FUNCTION_BLOCK Scanner_FB
VAR_INPUT
	mxEnable: BOOL;
	mxRP: BOOL;
	mxYP: BOOL;
	mxBP: BOOL;
	mxRCy: BOOL;
	mxYCy: BOOL;
	mxBCy: BOOL;
	mxYOct: BOOL;
	mxBOct: BOOL;
	mxROct: BOOL;
	mxIP: BOOL;
	mxRCon: BOOL;
	mxYCon: BOOL;
	mxBCon: BOOL;
END_VAR
VAR_OUTPUT
	
END_VAR
VAR
	TASK: INT;
	qxScanBuffer_1:BOOL;
	qxScanBuffer_2:BOOL;
	qxScanBuffer_3:BOOL;
	qxScanContainer:BOOL;
	mxPlate: BOOL;
	mxCylinder: BOOL;
	mxOctagon: BOOL;
	mxPART2: BOOL;
	mxPART3: BOOL;
	mxPart1: BOOL;
	mxSLOT1: BOOL;
	mxSLOT2: BOOL;
END_VAR

CASE TASK OF
	0:
	
		MAIN.ixAutoLamp:=FALSE;
		MAIN.ixManualLamp:=FALSE;
		MAIN.qxABBErrorLamp:=FALSE;
		MAIN.qxABBExecutLamp:=FALSE;
	
		IF ABB_Control_FB.Auto_Mode.Q1 THEN
			GVL.mwStationStatus:=0;
			IF GVL.BufferProducts.Storage1.Quatity>0 THEN
				TASK:=2;
			ELSE
				TASK:=1;
			END_IF
		ELSIF ABB_Control_FB.Manual_Mode.Q1 THEN
			GVL.mwStationStatus:=400;
			TASK:=1000;
		ELSIF GVL.ixEmergencyStop THEN 
						MAIN.qxEmergySTLamp:=TRUE;
						GVL.mwStationStatus:=1000;
						TASK:=2001;
		END_IF
	
	// AUTO MODE
	
	// Buffers Scanning
	1:
		GVL.mwStationStatus:=0;
		MAIN.qxABBExecutLamp:=TRUE;
		ABB_Control_FB.qxScanBuffer_1:=TRUE;
		ABB_Control_FB.mxScan:=TRUE;
		MAIN.qsTask:='Scan buffers';
		MAIN.qsSubTask:='Scan buffer 1';
	
		IF mxEnable THEN
			IF mxRP THEN
				GVL.BufferProducts.Storage1.Component:= 'Red Plate';
				GVL.BufferProducts.Storage1.Quatity:=2;
			ELSIF mxYP THEN
				GVL.BufferProducts.Storage1.Component:= 'Yellow Plate';
				GVL.BufferProducts.Storage1.Quatity:=2;
			ELSIF mxBP THEN
				GVL.BufferProducts.Storage1.Component:='Blue Plate';
				GVL.BufferProducts.Storage1.Quatity:=2;
			ELSIF mxRCy THEN
				GVL.BufferProducts.Storage1.Component:= 'Red Cylinder';
				GVL.BufferProducts.Storage1.Quatity:=4;
			ELSIF mxYCy THEN
				GVL.BufferProducts.Storage1.Component:= 'Yellow Cylinder';
				GVL.BufferProducts.Storage1.Quatity:=4;
			ELSIF mxBCy THEN
				GVL.BufferProducts.Storage1.Component:= 'Blue Cylinder';
				GVL.BufferProducts.Storage1.Quatity:=4;
			ELSIF mxROct THEN
				GVL.BufferProducts.Storage1.Component:= 'Red Octagon';
				GVL.BufferProducts.Storage1.Quatity:=4;
			ELSIF mxYOct THEN
				GVL.BufferProducts.Storage1.Component:= 'Yellow Octagon';
				GVL.BufferProducts.Storage1.Quatity:=4;
			ELSIF mxBOct THEN
				GVL.BufferProducts.Storage1.Component:= 'Blue Octagon';
				GVL.BufferProducts.Storage1.Quatity:=4;
			ELSIF mxIP THEN
				GVL.BufferProducts.Storage1.Component:='InvalidPart';
				GVL.BufferProducts.Storage1.Quatity:=0;
			END_IF
		END_IF
		
		IF GVL.BufferProducts.Storage1.Quatity=0 OR GVL.BufferProducts.Storage2.Quatity=0 OR GVL.BufferProducts.Storage3.Quatity=0 THEN
			MAIN.ixEmptyBuffer:=TRUE;
		ELSE
			MAIN.ixEmptyBuffer:=FALSE;
		END_IF
		
		IF ABB_Control_FB.mxBuffer_1_scanned THEN
			TASK:=2;
		END_IF
		
		IF
			GVL.ixEmergencyStop THEN 
						MAIN.qxEmergySTLamp:=TRUE;
						GVL.mwStationStatus:=1000;
						TASK:=2001;
		END_IF
	
	2:
		GVL.mwStationStatus:=0;
		MAIN.qxABBExecutLamp:=TRUE;
		ABB_Control_FB.mxScan:=FALSE;
		ABB_Control_FB.qxScanBuffer_1:=FALSE;
		IF GVL.BufferProducts.Storage2.Quatity>0 THEN
			TASK:=3;
		ELSE
			TASK:=4;
		END_IF
		
	4:
		GVL.mwStationStatus:=0;
		MAIN.qxABBExecutLamp:=TRUE;
		ABB_Control_FB.mxScan:=TRUE;
		ABB_Control_FB.qxScanBuffer_2:=TRUE;
		MAIN.qsTask:='Scan buffers';
		MAIN.qsSubTask:='Scan buffer 2';
			
		IF mxEnable THEN
			IF mxRP THEN
				GVL.BufferProducts.Storage2.Component:= 'Red Plate';
				GVL.BufferProducts.Storage2.Quatity:=2;
			ELSIF mxYP THEN
				GVL.BufferProducts.Storage2.Component:= 'Yellow Plate';
				GVL.BufferProducts.Storage2.Quatity:=2;
			ELSIF mxBP THEN
				GVL.BufferProducts.Storage2.Component:='Blue Plate';
				GVL.BufferProducts.Storage2.Quatity:=2;
			ELSIF mxRCy THEN
				GVL.BufferProducts.Storage2.Component:= 'Red Cylinder';
				GVL.BufferProducts.Storage2.Quatity:=4;
			ELSIF mxYCy THEN
				GVL.BufferProducts.Storage2.Component:= 'Yellow Cylinder';
				GVL.BufferProducts.Storage2.Quatity:=4;
			ELSIF mxBCy THEN
				GVL.BufferProducts.Storage2.Component:= 'Blue Cylinder';
				GVL.BufferProducts.Storage2.Quatity:=4;
			ELSIF mxROct THEN
				GVL.BufferProducts.Storage2.Component:= 'Red Octagon';
				GVL.BufferProducts.Storage2.Quatity:=4;
			ELSIF mxYOct THEN
				GVL.BufferProducts.Storage2.Component:= 'Yellow Octagon';
				GVL.BufferProducts.Storage2.Quatity:=4;
			ELSIF mxBOct THEN
				GVL.BufferProducts.Storage2.Component:= 'Blue Octagon';
				GVL.BufferProducts.Storage2.Quatity:=4;
			ELSIF mxIP THEN
				GVL.BufferProducts.Storage2.Component:='InvalidPart';
				GVL.BufferProducts.Storage2.Quatity:=0;
			END_IF
		END_IF
		
		IF GVL.BufferProducts.Storage1.Quatity=0 OR GVL.BufferProducts.Storage2.Quatity=0 OR GVL.BufferProducts.Storage3.Quatity=0 THEN
			MAIN.ixEmptyBuffer:=TRUE;
		ELSE
			MAIN.ixEmptyBuffer:=FALSE;
		END_IF
		
		IF ABB_Control_FB.mxBuffer_2_scanned THEN
			TASK:=3;
		END_IF
		
		IF
			GVL.ixEmergencyStop THEN 
						MAIN.qxEmergySTLamp:=TRUE;
						GVL.mwStationStatus:=1000;
						TASK:=2001;
		END_IF
		
	3:
		GVL.mwStationStatus:=0;
		MAIN.qxABBExecutLamp:=TRUE;
		ABB_Control_FB.mxScan:=FALSE;
		ABB_Control_FB.qxScanBuffer_2:=FALSE;
		IF GVL.BufferProducts.Storage3.Quatity>0 THEN
			TASK:=5;
		ELSE
			TASK:=6;
		END_IF
	
	6:
		GVL.mwStationStatus:=0;
		MAIN.qxABBExecutLamp:=TRUE;
		ABB_Control_FB.mxScan:=TRUE;
		ABB_Control_FB.qxScanBuffer_3:=TRUE;
		MAIN.qsTask:='Scan buffers';
		MAIN.qsSubTask:='Scan buffer 3';
		
		IF mxEnable THEN
			IF mxRP THEN
				GVL.BufferProducts.Storage3.Component:= 'Red Plate';
				GVL.BufferProducts.Storage3.Quatity:=2;
			ELSIF mxYP THEN
				GVL.BufferProducts.Storage3.Component:= 'Yellow Plate';
				GVL.BufferProducts.Storage3.Quatity:=2;
			ELSIF mxBP THEN
				GVL.BufferProducts.Storage3.Component:='Blue Plate';
				GVL.BufferProducts.Storage3.Quatity:=2;
			ELSIF mxRCy THEN
				GVL.BufferProducts.Storage3.Component:= 'Red Cylinder';
				GVL.BufferProducts.Storage3.Quatity:=4;
			ELSIF mxYCy THEN
				GVL.BufferProducts.Storage3.Component:= 'Yellow Cylinder';
				GVL.BufferProducts.Storage3.Quatity:=4;
			ELSIF mxBCy THEN
				GVL.BufferProducts.Storage3.Component:= 'Blue Cylinder';
				GVL.BufferProducts.Storage3.Quatity:=4;
			ELSIF mxROct THEN
				GVL.BufferProducts.Storage3.Component:= 'Red Octagon';
				GVL.BufferProducts.Storage3.Quatity:=4;
			ELSIF mxYOct THEN
				GVL.BufferProducts.Storage3.Component:= 'Yellow Octagon';
				GVL.BufferProducts.Storage3.Quatity:=4;
			ELSIF mxBOct THEN
				GVL.BufferProducts.Storage3.Component:= 'Blue Octagon';
				GVL.BufferProducts.Storage3.Quatity:=4;
			ELSIF mxIP THEN
				GVL.BufferProducts.Storage3.Component:='InvalidPart';
				GVL.BufferProducts.Storage3.Quatity:=0;
			END_IF
		END_IF
		
		IF GVL.BufferProducts.Storage1.Quatity=0 OR GVL.BufferProducts.Storage2.Quatity=0 OR GVL.BufferProducts.Storage3.Quatity=0 THEN
			MAIN.ixEmptyBuffer:=TRUE;
		ELSE
			MAIN.ixEmptyBuffer:=FALSE;
		END_IF
		
		IF ABB_Control_FB.mxBuffer_3_scanned THEN
			TASK:=5;
		END_IF
		
		IF
			GVL.ixEmergencyStop THEN 
						MAIN.qxEmergySTLamp:=TRUE;
						GVL.mwStationStatus:=1000;
						TASK:=2001;
		END_IF
		
	5:
		GVL.mwStationStatus:=0;
		MAIN.qxABBExecutLamp:=TRUE;
		ABB_Control_FB.mxScan:=FALSE;
		ABB_Control_FB.qxScanBuffer_3:=FALSE;
		TASK:=7;
		
	7:
		MAIN.qxABBExecutLamp:=FALSE;
		ABB_Control_FB.ixGoTo_AGV:=FALSE;
		ABB_Control_FB.qxAssemblyDone:=FALSE;
		GVL.qxPalletPlacedinAGV:=FALSE;
		ABB_Control_FB.mxConLeave:=FALSE;
		GVL.mwStationStatus:=100;
		IF GVL.BufferProducts.Storage1.Quatity>0 AND GVL.BufferProducts.Storage2.Quatity>0 AND GVL.BufferProducts.Storage3.Quatity>0 THEN
			TASK:=8;
		ELSE
			TASK:=0;
		END_IF
	
	8: // Containers Scanning
		MAIN.qsTask:='Waiting for AGV';
		MAIN.qsSubTask:='';
		
		IF GVL.ixAGVatStation THEN
			GVL.mwStationStatus:=300;
			MAIN.qxABBExecutLamp:=TRUE;
			ABB_Control_FB.ixGoTo_AGV:=TRUE;
			ABB_Control_FB.mxScan:= TRUE;
			MAIN.qsTask:='Go to AGV Pos';
			MAIN.qsSubTask:='Pick Container';
			
			IF ABB_Control_FB.ABBPickLeaveContainerAGVPick_1.mxDone THEN
				MAIN.qsTask:='Go to Scanner';
				MAIN.qsSubTask:='Scanning Container';
			END_IF
			
			IF mxEnable THEN
				IF mxRCon THEN
					MAIN.qsContainer:='Red Container';
				ELSIF mxYCon THEN
					MAIN.qsContainer:='Yellow Container';
				ELSIF mxBCon THEN
					MAIN.qsContainer:='Blue Container';
				END_IF
				TASK:=9;
			END_IF
		END_IF
	
	9: // Parts Scanning
		IF ABB_Control_FB.mxContainerScanDone THEN
			TASK:=44;
		END_IF
		
		IF
			GVL.ixEmergencyStop THEN 
						MAIN.qxEmergySTLamp:=TRUE;
						GVL.mwStationStatus:=1000;
						TASK:=2001;
		END_IF
		
	44:
	
		ABB_Control_FB.ixGoTo_AGV:=FALSE;
		ABB_Control_FB.qxCon1:=TRUE;
		MAIN.qsTask:='Scan Products on Container';
		MAIN.qsSubTask:='Scan Plate';
		IF ABB_Control_FB.mxCon_1_ATtableScan THEN
			IF GVL.ixInductiveSensorinTool THEN
				MAIN.mxPlateAvailable:=TRUE;
				TASK:=10;
			ELSIF NOT GVL.ixInductiveSensorinTool THEN
				TASK:=100;
			END_IF
		END_IF
		
	10:
		ABB_Control_FB.mxCon_1_ATtableScan:=FALSE;
		ABB_Control_FB.qxCon1:=FALSE;
		TASK:=11;
		
	11:
		ABB_Control_FB.qxCon2:=TRUE;
		MAIN.qsTask:='Scan Products on Container';
		MAIN.qsSubTask:='Scan Cylinder';
		IF ABB_Control_FB.mxCon_2_ATtableScan THEN
			IF GVL.ixInductiveSensorinTool THEN
				MAIN.mxCylinderAvailable:=TRUE;
				TASK:=12;
			ELSIF NOT GVL.ixInductiveSensorinTool THEN
				TASK:=101;
			END_IF
		END_IF
		
	12:
		ABB_Control_FB.mxCon_2_ATtableScan:=FALSE;
		ABB_Control_FB.qxCon2:=FALSE;
		TASK:=13;
		
	13:
		ABB_Control_FB.qxCon3:=TRUE;
		MAIN.qsTask:='Scan Products on Container';
		MAIN.qsSubTask:='Scan Octagon';
		IF ABB_Control_FB.mxCon_3_ATtableScan THEN
			IF GVL.ixInductiveSensorinTool THEN
				MAIN.mxOctagonAvailable:=TRUE;
				TASK:=350;
			ELSIF NOT GVL.ixInductiveSensorinTool THEN
				TASK:=102;
			END_IF
		END_IF
		
	100:
		GVL.ixAGVatStation:=FALSE;
		ABB_Control_FB.qxCon1:=FALSE;
		
		IF MAIN.qsContainer='Red Container' THEN
			IF GVL.BufferProducts.Storage1.Component='Red Plate' AND GVL.BufferProducts.Storage1.Quatity>0 THEN
				MAIN.mwBufferID:=1;
				ABB_Control_FB.qxPart_1_Assemble:=TRUE;
				MAIN.qsTask:='Assembly';
				MAIN.qsSubTask:='Assembling Red Plate';
				GVL.BufferProducts.Storage1.Quatity:=GVL.BufferProducts.Storage1.Quatity-1;
				TASK:=200;
			ELSIF GVL.BufferProducts.Storage2.Component='Red Plate' AND GVL.BufferProducts.Storage2.Quatity>0 THEN
				MAIN.mwBufferID:=2;
				ABB_Control_FB.qxPart_2_Assemble:=TRUE;
				MAIN.qsTask:='Assembly';
				MAIN.qsSubTask:='Assembling Red Plate';
				GVL.BufferProducts.Storage2.Quatity:=GVL.BufferProducts.Storage2.Quatity-1;
				TASK:=200;
			ELSIF GVL.BufferProducts.Storage3.Component='Red Plate' AND GVL.BufferProducts.Storage3.Quatity>0 THEN
				MAIN.mwBufferID:=3;
				ABB_Control_FB.qxPart_3_Assemble:=TRUE;
				MAIN.qsTask:='Assembly';
				MAIN.qsSubTask:='Assembling Red Plate';
				GVL.BufferProducts.Storage3.Quatity:=GVL.BufferProducts.Storage3.Quatity-1;
				TASK:=200;
			ELSE
				TASK:=150;				
			END_IF
			
		ELSIF MAIN.qsContainer='Yellow Container' THEN
			IF GVL.BufferProducts.Storage1.Component='Yellow Plate' AND GVL.BufferProducts.Storage1.Quatity>0 THEN
				MAIN.mwBufferID:=1;
				ABB_Control_FB.qxPart_1_Assemble:=TRUE;
				MAIN.qsTask:='Assembly';
				MAIN.qsSubTask:='Assembling Yellow Plate';
				GVL.BufferProducts.Storage1.Quatity:=GVL.BufferProducts.Storage1.Quatity-1;
				TASK:=200;
			ELSIF GVL.BufferProducts.Storage2.Component='Yellow Plate' AND GVL.BufferProducts.Storage2.Quatity>0 THEN
				MAIN.mwBufferID:=2;
				ABB_Control_FB.qxPart_2_Assemble:=TRUE;
				MAIN.qsTask:='Assembly';
				MAIN.qsSubTask:='Assembling Yellow Plate';
				GVL.BufferProducts.Storage2.Quatity:=GVL.BufferProducts.Storage2.Quatity-1;
				TASK:=200;
			ELSIF GVL.BufferProducts.Storage3.Component='Yellow Plate' AND GVL.BufferProducts.Storage3.Quatity>0 THEN
				MAIN.mwBufferID:=3;
				ABB_Control_FB.qxPart_3_Assemble:=TRUE;
				MAIN.qsTask:='Assembly';
				MAIN.qsSubTask:='Assembling Yellow Plate';
				GVL.BufferProducts.Storage3.Quatity:=GVL.BufferProducts.Storage3.Quatity-1;
				TASK:=200;
			ELSE
				TASK:=150;
			END_IF
			
		ELSIF MAIN.qsContainer='Blue Container' THEN
			IF GVL.BufferProducts.Storage1.Component='Blue Plate' AND GVL.BufferProducts.Storage1.Quatity>0 THEN
				MAIN.mwBufferID:=1;
				ABB_Control_FB.qxPart_1_Assemble:=TRUE;
				MAIN.qsTask:='Assembly';
				MAIN.qsSubTask:='Assembling Blue Plate';
				GVL.BufferProducts.Storage1.Quatity:=GVL.BufferProducts.Storage1.Quatity-1;
				TASK:=200;
			ELSIF GVL.BufferProducts.Storage2.Component='Blue Plate' AND GVL.BufferProducts.Storage2.Quatity>0 THEN
				MAIN.mwBufferID:=2;
				ABB_Control_FB.qxPart_2_Assemble:=TRUE;
				MAIN.qsTask:='Assembly';
				MAIN.qsSubTask:='Assembling Blue Plate';
				GVL.BufferProducts.Storage2.Quatity:=GVL.BufferProducts.Storage2.Quatity-1;
				TASK:=200;
			ELSIF GVL.BufferProducts.Storage3.Component='Blue Plate' AND GVL.BufferProducts.Storage3.Quatity>0 THEN
				MAIN.mwBufferID:=3;
				ABB_Control_FB.qxPart_3_Assemble:=TRUE;
				MAIN.qsTask:='Assembly';
				MAIN.qsSubTask:='Assembling Blue Plate';
				GVL.BufferProducts.Storage3.Quatity:=GVL.BufferProducts.Storage3.Quatity-1;
				TASK:=200;
			ELSE
				TASK:=150;
			END_IF		
		END_IF
		
		IF
			GVL.ixEmergencyStop THEN 
						MAIN.qxEmergySTLamp:=TRUE;
						GVL.mwStationStatus:=1000;
						TASK:=2001;
		END_IF
	
	200:
		IF ABB_Control_FB.mxAsse_1_done THEN
			MAIN.qsTask:='Assembly';
			MAIN.qsSubTask:='Plate Assembled';
			MAIN.mxPlateAvailable:=TRUE;
			mxPlate:=TRUE;
			ABB_Control_FB.qxPart_1_Assemble:=FALSE;
			TASK:=10;
		ELSIF ABB_Control_FB.mxAsse_2_done THEN
			MAIN.qsTask:='Assembly';
			MAIN.qsSubTask:='Plate Assembled';
			MAIN.mxPlateAvailable:=TRUE;
			mxPlate:=TRUE;
			ABB_Control_FB.qxPart_2_Assemble:=FALSE;
			TASK:=10;
		ELSIF ABB_Control_FB.mxAsse_3_done THEN
			MAIN.qsTask:='Assembly';
			MAIN.qsSubTask:='Plate Assembled';
			MAIN.mxPlateAvailable:=TRUE;
			mxPlate:=TRUE;
			ABB_Control_FB.qxPart_3_Assemble:=FALSE;
			TASK:=10;
		END_IF
		
	101:
		IF MAIN.qsContainer='Red Container' THEN
			IF GVL.BufferProducts.Storage1.Component='Red Cylinder' AND GVL.BufferProducts.Storage1.Quatity>0 THEN
				MAIN.mwBufferID:=1;
				ABB_Control_FB.qxPart_1_Assemble:=TRUE;
				MAIN.qsTask:='Assembly';
				MAIN.qsSubTask:='Assembling Red Cylinder';
				GVL.BufferProducts.Storage1.Quatity:=GVL.BufferProducts.Storage1.Quatity-1;
				TASK:=201;
			ELSIF GVL.BufferProducts.Storage2.Component='Red Cylinder' AND GVL.BufferProducts.Storage2.Quatity>0 THEN
				MAIN.mwBufferID:=2;
				ABB_Control_FB.qxPart_2_Assemble:=TRUE;
				MAIN.qsTask:='Assembly';
				MAIN.qsSubTask:='Assembling Red Cylinder';
				GVL.BufferProducts.Storage2.Quatity:=GVL.BufferProducts.Storage2.Quatity-1;
				TASK:=201;
			ELSIF GVL.BufferProducts.Storage3.Component='Red Cylinder' AND GVL.BufferProducts.Storage3.Quatity>0 THEN
				MAIN.mwBufferID:=3;
				ABB_Control_FB.qxPart_3_Assemble:=TRUE;
				MAIN.qsTask:='Assembly';
				MAIN.qsSubTask:='Assembling Red Cylinder';
				GVL.BufferProducts.Storage3.Quatity:=GVL.BufferProducts.Storage3.Quatity-1;
				TASK:=201;
			ELSE
				TASK:=12;				
			END_IF
			
		ELSIF MAIN.qsContainer='Yellow Container' THEN
			IF GVL.BufferProducts.Storage1.Component='Yellow Cylinder' AND GVL.BufferProducts.Storage1.Quatity>0 THEN
				MAIN.mwBufferID:=1;
				ABB_Control_FB.qxPart_1_Assemble:=TRUE;
				MAIN.qsTask:='Assembly';
				MAIN.qsSubTask:='Assembling Yellow Cylinder';
				GVL.BufferProducts.Storage1.Quatity:=GVL.BufferProducts.Storage1.Quatity-1;
				TASK:=201;
			ELSIF GVL.BufferProducts.Storage2.Component='Yellow Cylinder' AND GVL.BufferProducts.Storage2.Quatity>0 THEN
				MAIN.mwBufferID:=2;
				ABB_Control_FB.qxPart_2_Assemble:=TRUE;
				MAIN.qsTask:='Assembly';
				MAIN.qsSubTask:='Assembling Yellow Cylinder';
				GVL.BufferProducts.Storage2.Quatity:=GVL.BufferProducts.Storage2.Quatity-1;
				TASK:=201;
			ELSIF GVL.BufferProducts.Storage3.Component='Yellow Cylinder' AND GVL.BufferProducts.Storage3.Quatity>0 THEN
				MAIN.mwBufferID:=3;
				ABB_Control_FB.qxPart_3_Assemble:=TRUE;
				MAIN.qsTask:='Assembly';
				MAIN.qsSubTask:='Assembling Yellow Cylinder';
				GVL.BufferProducts.Storage3.Quatity:=GVL.BufferProducts.Storage3.Quatity-1;
				TASK:=201;
			ELSE
				TASK:=12;
			END_IF
			
		ELSIF MAIN.qsContainer='Blue Container' THEN
			IF GVL.BufferProducts.Storage1.Component='Blue Cylinder' AND GVL.BufferProducts.Storage1.Quatity>0 THEN
				MAIN.mwBufferID:=1;
				ABB_Control_FB.qxPart_1_Assemble:=TRUE;
				MAIN.qsTask:='Assembly';
				MAIN.qsSubTask:='Assembling Blue Cylinder';
				GVL.BufferProducts.Storage1.Quatity:=GVL.BufferProducts.Storage1.Quatity-1;
				TASK:=201;
			ELSIF GVL.BufferProducts.Storage2.Component='Blue Cylinder' AND GVL.BufferProducts.Storage2.Quatity>0 THEN
				MAIN.mwBufferID:=2;
				ABB_Control_FB.qxPart_2_Assemble:=TRUE;
				MAIN.qsTask:='Assembly';
				MAIN.qsSubTask:='Assembling Blue Cylinder';
				GVL.BufferProducts.Storage2.Quatity:=GVL.BufferProducts.Storage2.Quatity-1;
				TASK:=201;
			ELSIF GVL.BufferProducts.Storage3.Component='Blue Cylinder' AND GVL.BufferProducts.Storage3.Quatity>0 THEN
				MAIN.mwBufferID:=3;
				ABB_Control_FB.qxPart_3_Assemble:=TRUE;
				MAIN.qsTask:='Assembly';
				MAIN.qsSubTask:='Assembling Blue Cylinder';
				GVL.BufferProducts.Storage3.Quatity:=GVL.BufferProducts.Storage3.Quatity-1;
				TASK:=201;
			ELSE
				TASK:=12;
			END_IF		
		END_IF
		
		IF
			GVL.ixEmergencyStop THEN 
						MAIN.qxEmergySTLamp:=TRUE;
						GVL.mwStationStatus:=1000;
						TASK:=2001;
		END_IF
		
	102:
		ABB_Control_FB.qxCon3:=FALSE;
		IF MAIN.qsContainer='Red Container' THEN
			IF GVL.BufferProducts.Storage1.Component='Red Octagon' AND GVL.BufferProducts.Storage1.Quatity>0 THEN
				MAIN.mwBufferID:=1;
				ABB_Control_FB.qxPart_1_Assemble:=TRUE;
				MAIN.qsTask:='Assembly';
				MAIN.qsSubTask:='Assembling Red Octagon';
				GVL.BufferProducts.Storage1.Quatity:=GVL.BufferProducts.Storage1.Quatity-1;
				TASK:=600;
			ELSIF GVL.BufferProducts.Storage2.Component='Red Octagon' AND GVL.BufferProducts.Storage2.Quatity>0 THEN
				MAIN.mwBufferID:=2;
				ABB_Control_FB.qxPart_2_Assemble:=TRUE;
				MAIN.qsTask:='Assembly';
				MAIN.qsSubTask:='Assembling Red Octagon';
				GVL.BufferProducts.Storage2.Quatity:=GVL.BufferProducts.Storage2.Quatity-1;
				TASK:=600;
			ELSIF GVL.BufferProducts.Storage3.Component='Red Octagon' AND GVL.BufferProducts.Storage3.Quatity>0 THEN
				MAIN.mwBufferID:=3;
				ABB_Control_FB.qxPart_3_Assemble:=TRUE;
				MAIN.qsTask:='Assembly';
				MAIN.qsSubTask:='Assembling Red Octagon';
				GVL.BufferProducts.Storage3.Quatity:=GVL.BufferProducts.Storage3.Quatity-1;
				TASK:=600;
			ELSE
				TASK:=350;				
			END_IF
			
		ELSIF MAIN.qsContainer='Yellow Container' THEN
			IF GVL.BufferProducts.Storage1.Component='Yellow Octagon' AND GVL.BufferProducts.Storage1.Quatity>0 THEN
				MAIN.mwBufferID:=1;
				ABB_Control_FB.qxPart_1_Assemble:=TRUE;
				MAIN.qsTask:='Assembly';
				MAIN.qsSubTask:='Assembling Yellow Octagon';
				GVL.BufferProducts.Storage1.Quatity:=GVL.BufferProducts.Storage1.Quatity-1;
				TASK:=600;
			ELSIF GVL.BufferProducts.Storage2.Component='Yellow Octagon' AND GVL.BufferProducts.Storage2.Quatity>0 THEN
				MAIN.mwBufferID:=2;
				ABB_Control_FB.qxPart_2_Assemble:=TRUE;
				MAIN.qsTask:='Assembly';
				MAIN.qsSubTask:='Assembling Yellow Octagon';
				GVL.BufferProducts.Storage2.Quatity:=GVL.BufferProducts.Storage2.Quatity-1;
				TASK:=600;
			ELSIF GVL.BufferProducts.Storage3.Component='Yellow Octagon' AND GVL.BufferProducts.Storage3.Quatity>0 THEN
				MAIN.mwBufferID:=3;
				ABB_Control_FB.qxPart_3_Assemble:=TRUE;
				MAIN.qsTask:='Assembly';
				MAIN.qsSubTask:='Assembling Yellow Octagon';
				GVL.BufferProducts.Storage3.Quatity:=GVL.BufferProducts.Storage3.Quatity-1;
				TASK:=600;
			ELSE
				TASK:=350;
			END_IF
			
		ELSIF MAIN.qsContainer='Blue Container' THEN
			IF GVL.BufferProducts.Storage1.Component='Blue Octagon' AND GVL.BufferProducts.Storage1.Quatity>0 THEN
				MAIN.mwBufferID:=1;
				ABB_Control_FB.qxPart_1_Assemble:=TRUE;
				MAIN.qsTask:='Assembly';
				MAIN.qsSubTask:='Assembling Blue Octagon';
				GVL.BufferProducts.Storage1.Quatity:=GVL.BufferProducts.Storage1.Quatity-1;
				TASK:=600;
			ELSIF GVL.BufferProducts.Storage2.Component='Blue Octagon' AND GVL.BufferProducts.Storage2.Quatity>0 THEN
				MAIN.mwBufferID:=2;
				ABB_Control_FB.qxPart_2_Assemble:=TRUE;
				MAIN.qsTask:='Assembly';
				MAIN.qsSubTask:='Assembling Blue Octagon';
				GVL.BufferProducts.Storage2.Quatity:=GVL.BufferProducts.Storage2.Quatity-1;
				TASK:=600;
			ELSIF GVL.BufferProducts.Storage3.Component='Blue Octagon' AND GVL.BufferProducts.Storage3.Quatity>0 THEN
				MAIN.mwBufferID:=3;
				ABB_Control_FB.qxPart_3_Assemble:=TRUE;
				MAIN.qsTask:='Assembly';
				MAIN.qsSubTask:='Assembling Blue Octagon';
				GVL.BufferProducts.Storage3.Quatity:=GVL.BufferProducts.Storage3.Quatity-1;
				TASK:=600;
			ELSE
				TASK:=350;
			END_IF		
		END_IF
		
		IF
			GVL.ixEmergencyStop THEN 
						MAIN.qxEmergySTLamp:=TRUE;
						GVL.mwStationStatus:=1000;
						TASK:=2001;
		END_IF
		
	201: 
		IF ABB_Control_FB.mxAsse_1_done THEN
			MAIN.qsTask:='Assembly';
			MAIN.qsSubTask:='Cylinder Assembled';
			MAIN.mxCylinderAvailable:=TRUE;
			ABB_Control_FB.qxPart_1_Assemble:=FALSE;
			TASK:=12;
		ELSIF ABB_Control_FB.mxAsse_2_done THEN
			MAIN.qsTask:='Assembly';
			MAIN.qsSubTask:='Cylinder Assembled';
			MAIN.mxCylinderAvailable:=TRUE;
			ABB_Control_FB.qxPart_2_Assemble:=FALSE;
			TASK:=12;
		ELSIF ABB_Control_FB.mxAsse_3_done THEN
			MAIN.qsTask:='Assembly';
			MAIN.qsSubTask:='Cylinder Assembled';
			MAIN.mxCylinderAvailable:=TRUE;
			ABB_Control_FB.qxPart_3_Assemble:=FALSE;
			TASK:=12;
		END_IF
	
	600:
		IF ABB_Control_FB.mxAsse_1_done THEN
			MAIN.qsTask:='Assembly';
			MAIN.qsSubTask:='Octagon Assembled';
			MAIN.mxOctagonAvailable:=TRUE;
			mxOctagon:=TRUE;
			ABB_Control_FB.qxPart_1_Assemble:=FALSE;
			TASK:=700;
		ELSIF ABB_Control_FB.mxAsse_2_done THEN
			MAIN.qsTask:='Assembly';
			MAIN.qsSubTask:='Octagon Assembled';
			MAIN.mxOctagonAvailable:=TRUE;
			mxOctagon:=TRUE;
			ABB_Control_FB.qxPart_2_Assemble:=FALSE;
			TASK:=700;
		ELSIF ABB_Control_FB.mxAsse_3_done THEN
			MAIN.qsTask:='Assembly';
			MAIN.qsSubTask:='Octagon Assembled';
			MAIN.mxOctagonAvailable:=TRUE;
			mxOctagon:=TRUE;
			ABB_Control_FB.qxPart_3_Assemble:=FALSE;
			TASK:=700;
		END_IF
		
	700:
		IF MAIN.mxPlateAvailable AND MAIN.mxCylinderAvailable AND MAIN.mxOctagonAvailable THEN
			ABB_Control_FB.qxAssemblyDone:=TRUE;
			GVL.qsOrderFornextAssembly:='Assembled Product';
			IF ABB_Control_FB.mxConLeave THEN
				MAIN.mxPlateAvailable:=FALSE;
				MAIN.mxCylinderAvailable:=FALSE;
				MAIN.mxOctagonAvailable:=FALSE;
				GVL.qxPalletPlacedinAGV:=TRUE;
				GVL.qsOrderFornextAssembly:='0';
				TASK:=7;
			END_IF
		END_IF
	
	150: // Order for Plates
		IF MAIN.qsContainer='Red Container' THEN
			GVL.qsOrderFornextAssembly:='Red Plate';
			TASK:=111;
		ELSIF MAIN.qsContainer='Yellow Container' THEN
			GVL.qsOrderFornextAssembly:='Yellow Plate';
			TASK:=111;
		ELSIF MAIN.qsContainer='Blue Container' THEN
			GVL.qsOrderFornextAssembly:='Blue Plate';
			TASK:=111;
		END_IF
		
	350: // Order for missing Parts
		ABB_Control_FB.qxCon3:=FALSE;
		ABB_Control_FB.qxPart_3_Assemble:=FALSE;
		
		IF mxCylinder OR MAIN.mxCylinderAvailable THEN
			mxPART2:=TRUE;
			TASK:=351;
		ELSE
			mxPART2:=FALSE;
			TASK:=351;
		END_IF
		
	351:
		IF mxOctagon OR MAIN.mxOctagonAvailable THEN
			mxPART3:=TRUE;
			TASK:=352;
		ELSE
			mxPART3:=FALSE;
			TASK:=352;
		END_IF
		
	352:
		IF MAIN.qsContainer='Red Container' THEN
			IF mxPART2 AND mxPART3 THEN
				GVL.qsOrderFornextAssembly:='Assembled Product';
				TASK:=111;
			ELSIF mxPART2 AND NOT mxPART3 THEN
				GVL.qsOrderFornextAssembly:='Red Octagon';
				TASK:=111;
			ELSIF NOT mxPART2 AND mxPART3 THEN
				GVL.qsOrderFornextAssembly:='Red Cylinder';
				TASK:=111;
			ELSIF NOT mxPART2 AND NOT mxPART3 THEN
				GVL.qsOrderFornextAssembly:='Red Cylinder';
				TASK:=111;
			END_IF
			
		ELSIF MAIN.qsContainer='Yellow Container' THEN
			IF mxPART2 AND mxPART3 THEN
				GVL.qsOrderFornextAssembly:='Assembled Product';
				TASK:=111;
			ELSIF mxPART2 AND NOT mxPART3 THEN
				GVL.qsOrderFornextAssembly:='Yellow Octagon';
				TASK:=111;
			ELSIF NOT mxPART2 AND mxPART3 THEN
				GVL.qsOrderFornextAssembly:='Yellow Cylinder';
				TASK:=111;
			ELSIF NOT mxPART2 AND NOT mxPART3 THEN
				GVL.qsOrderFornextAssembly:='Yellow Cylinder';
				TASK:=111;
			END_IF
			
		ELSIF MAIN.qsContainer='Blue Container' THEN
			IF mxPART2 AND mxPART3 THEN
				GVL.qsOrderFornextAssembly:='Assembled Product';
				TASK:=111;
			ELSIF mxPART2 AND NOT mxPART3 THEN
				GVL.qsOrderFornextAssembly:='Blue Octagon';
				TASK:=111;
			ELSIF NOT mxPART2 AND mxPART3 THEN
				GVL.qsOrderFornextAssembly:='Blue Cylinder';
				TASK:=111;
			ELSIF NOT mxPART2 AND NOT mxPART3 THEN
				GVL.qsOrderFornextAssembly:='Blue Cylinder';
				TASK:=111;
			END_IF
		END_IF
		
		
	111:
		ABB_Control_FB.qxPart_1_Assemble:=FALSE;
		ABB_Control_FB.qxPart_2_Assemble:=FALSE;
		ABB_Control_FB.qxPart_3_Assemble:=FALSE;
		ABB_Control_FB.qxCon1:=FALSE;
		ABB_Control_FB.qxCon2:=FALSE;
		ABB_Control_FB.qxCon3:=FALSE;
		ABB_Control_FB.ixGoTo_AGV:=FALSE;
		ABB_Control_FB.qxScanBuffer_1:=FALSE;
		ABB_Control_FB.qxScanBuffer_2:=FALSE;
		ABB_Control_FB.qxScanBuffer_3:=FALSE;
		mxPART2:=FALSE;
		mxPART3:=FALSE;
		ABB_Control_FB.qxAssemblyDone:=TRUE;
		GVL.qsOrderFornextAssembly:='Assembled Product';
		IF ABB_Control_FB.ABBGotoAGVPos_Assembled.mxEnable THEN
			MAIN.qsTask:='Go to AGV Pos';
			MAIN.qsSubTask:='Leave Container';
			TASK:=121;
		END_IF
		
	121:
		IF ABB_Control_FB.mxConLeave THEN
			mxPlate:=FALSE;
			mxCylinder:=FALSE;
			mxOctagon:=FALSE;
			MAIN.mxPlateAvailable:=FALSE;
			MAIN.mxCylinderAvailable:=FALSE;
			MAIN.mxOctagonAvailable:=FALSE;
			GVL.qxPalletPlacedinAGV:=TRUE;
			GVL.qsOrderFornextAssembly:='0';
			MAIN.qsContainer:='';
			TASK:=7;
		END_IF
		
		
	// MANUAL MODE
	
	1000:
		GVL.mwStationStatus:=400;
		IF ABB_Control_FB.ixGotoHome THEN
			ABB_Control_FB.qxGotoHome:=TRUE;
			MAIN.qxABBExecutLamp:=TRUE;
			TASK:=1100;
		ELSIF ABB_Control_FB.ixGotoAGV THEN
			ABB_Control_FB.qxGotoAGV:=TRUE;
			MAIN.qxABBExecutLamp:=TRUE;
			TASK:=1200;
		ELSIF ABB_Control_FB.ixGotoTable THEN
			ABB_Control_FB.qxGotoTable:=TRUE;
			MAIN.qxABBExecutLamp:=TRUE;
			TASK:=1300;
		ELSIF ABB_Control_FB.ixGotoBuffer THEN
			ABB_Control_FB.qxGotoBuffer:=TRUE;
			MAIN.qxABBExecutLamp:=TRUE;
			TASK:=1400;
		ELSIF ABB_Control_FB.ixGotoScanner THEN
			ABB_Control_FB.qxGotoScanner:=TRUE;
			MAIN.qxABBExecutLamp:=TRUE;
			TASK:=1500;
		ELSIF ABB_Control_FB.ixPickBuffer1 THEN
			ABB_Control_FB.qxPickBuffer1:=TRUE;
			MAIN.qxABBExecutLamp:=TRUE;
			TASK:=1600;
		ELSIF ABB_Control_FB.ixLeaveBuffer1 THEN
			ABB_Control_FB.qxLeaveBuffer1:=TRUE;
			MAIN.qxABBExecutLamp:=TRUE;
			TASK:=1700;
		ELSIF ABB_Control_FB.ixPickBuffer2 THEN
			ABB_Control_FB.qxPickBuffer2:=TRUE;
			MAIN.qxABBExecutLamp:=TRUE;
			TASK:=1600;
		ELSIF ABB_Control_FB.ixLeaveBuffer2 THEN
			ABB_Control_FB.qxLeaveBuffer2:=TRUE;
			MAIN.qxABBExecutLamp:=TRUE;
			TASK:=1700;
		ELSIF ABB_Control_FB.ixPickBuffer3 THEN
			ABB_Control_FB.qxPickBuffer3:=TRUE;
			MAIN.qxABBExecutLamp:=TRUE;
			TASK:=1600;
		ELSIF ABB_Control_FB.ixLeaveBuffer3 THEN
			ABB_Control_FB.qxLeaveBuffer3:=TRUE;
			MAIN.qxABBExecutLamp:=TRUE;
			TASK:=1700;
		ELSIF ABB_Control_FB.ixPickScanner THEN
			ABB_Control_FB.qxPickScanner:=TRUE;
			MAIN.qxABBExecutLamp:=TRUE;
			TASK:=1800;
		ELSIF ABB_Control_FB.ixLeaveScanner THEN
			ABB_Control_FB.qxLeaveScanner:=TRUE;
			MAIN.qxABBExecutLamp:=TRUE;
			TASK:=1900;
		ELSIF ABB_Control_FB.ixPickAGV THEN
			ABB_Control_FB.qxPickAGV:=TRUE;
			MAIN.qxABBExecutLamp:=TRUE;
			TASK:=2000;
		ELSIF ABB_Control_FB.ixLeaveAGV THEN
			ABB_Control_FB.qxLeaveAGV:=TRUE;
			MAIN.qxABBExecutLamp:=TRUE;
			TASK:=2100;
		ELSIF ABB_Control_FB.ixPickTable THEN
			ABB_Control_FB.qxPickTable:=TRUE;
			MAIN.qxABBExecutLamp:=TRUE;
			TASK:=2500;
		ELSIF ABB_Control_FB.ixLeaveTable THEN
			ABB_Control_FB.qxLeaveTable:=TRUE;
			MAIN.qxABBExecutLamp:=TRUE;
			TASK:=2600;
		ELSIF ABB_Control_FB.ixScanBuffer THEN
			ABB_Control_FB.mxScan:=TRUE;
			IF MAIN.mwBufferID=1 THEN
				TASK:=2200;
			ELSIF MAIN.mwBufferID=2 THEN
				TASK:=2300;
			ELSIF MAIN.mwBufferID=3 THEN
				TASK:=2400;
			END_IF
		ELSIF ABB_Control_FB.ixScanContainer THEN
			ABB_Control_FB.mxScan:=TRUE;
			TASK:=2700;
		ELSIF ABB_Control_FB.ixScanPart1 THEN
			MAIN.qxABBExecutLamp:=TRUE;
			TASK:=2800;
		ELSIF ABB_Control_FB.ixScanPart2 THEN
			MAIN.qxABBExecutLamp:=TRUE;
			TASK:=2900;
		ELSIF ABB_Control_FB.ixScanPart3 THEN
			MAIN.qxABBExecutLamp:=TRUE;
			TASK:=3000;
		ELSIF ABB_Control_FB.ixAssemble1 THEN
			MAIN.qxABBExecutLamp:=TRUE;
			GVL.BufferProducts.Storage1.Quatity:=GVL.BufferProducts.Storage1.Quatity-1;
			TASK:=3100;
		ELSIF ABB_Control_FB.ixAssemble2 THEN
			MAIN.qxABBExecutLamp:=TRUE;
			GVL.BufferProducts.Storage2.Quatity:=GVL.BufferProducts.Storage2.Quatity-1;
			TASK:=3200;
		ELSIF ABB_Control_FB.ixAssemble3 THEN
			MAIN.qxABBExecutLamp:=TRUE;
			GVL.BufferProducts.Storage3.Quatity:=GVL.BufferProducts.Storage3.Quatity-1;
			TASK:=3300;
		ELSIF ABB_Control_FB.ixSendOrder THEN
			TASK:=3400;
		ELSIF ABB_Control_FB.ixFinishOrder THEN
			TASK:=3900;
			
		END_IF
		
	1100:
		IF ABB_Control_FB.qxHOME THEN
			MAIN.qxABBExecutLamp:=FALSE;
			ABB_Control_FB.qxGotoHome:=FALSE;
			ABB_Control_FB.ixGotoHome:=FALSE;
			TASK:=1000;
		END_IF
		
	1200:
		IF ABB_Control_FB.qxAGV THEN
			MAIN.qxABBExecutLamp:=FALSE;
			ABB_Control_FB.qxGotoAGV:=FALSE;
			ABB_Control_FB.ixGotoAGV:=FALSE;
			TASK:=1000;
		END_IF
		
	1300:
		IF ABB_Control_FB.qxTABLE THEN
			MAIN.qxABBExecutLamp:=FALSE;
			ABB_Control_FB.qxGotoTable:=FALSE;
			ABB_Control_FB.ixGotoTable:=FALSE;
			TASK:=1000;
		END_IF
		
	1400:
		IF ABB_Control_FB.qxBUFFER THEN
			MAIN.qxABBExecutLamp:=FALSE;
			ABB_Control_FB.qxGotoBuffer:=FALSE;
			ABB_Control_FB.ixGotoBuffer:=FALSE;
			TASK:=1000;
		END_IF
		
	1500:
		IF ABB_Control_FB.qxSCANNER THEN
			MAIN.qxABBExecutLamp:=FALSE;
			ABB_Control_FB.qxGotoScanner:=FALSE;
			ABB_Control_FB.ixGotoScanner:=FALSE;
			TASK:=1000;
		END_IF
		
	1600:
		IF ABB_Control_FB.qxBufferPicked1 THEN
			MAIN.qxABBExecutLamp:=FALSE;
			ABB_Control_FB.qxPickBuffer1:=FALSE;
			ABB_Control_FB.ixPickBuffer1:=FALSE;
			ABB_Control_FB.qxPickBuffer2:=FALSE;
			ABB_Control_FB.ixPickBuffer2:=FALSE;
			ABB_Control_FB.qxPickBuffer3:=FALSE;
			ABB_Control_FB.ixPickBuffer3:=FALSE;
			TASK:=1000;
		END_IF
		
	1700:
		IF ABB_Control_FB.qxBufferLeft1 THEN
			MAIN.qxABBExecutLamp:=FALSE;
			ABB_Control_FB.qxPickBuffer1:=FALSE;
			ABB_Control_FB.ixPickBuffer1:=FALSE;
			ABB_Control_FB.qxPickBuffer2:=FALSE;
			ABB_Control_FB.ixPickBuffer2:=FALSE;
			ABB_Control_FB.qxPickBuffer3:=FALSE;
			ABB_Control_FB.ixPickBuffer3:=FALSE;
			TASK:=1000;
		END_IF
		
	1800:
		IF ABB_Control_FB.qxPickedScanner THEN
			MAIN.qxABBExecutLamp:=FALSE;
			ABB_Control_FB.qxPickScanner:=FALSE;
			ABB_Control_FB.ixPickScanner:=FALSE;
			TASK:=1000;
		END_IF
		
	1900:
		IF ABB_Control_FB.qxLeftScanner THEN
			MAIN.qxABBExecutLamp:=FALSE;
			ABB_Control_FB.qxLeaveScanner:=FALSE;
			ABB_Control_FB.ixLeaveScanner:=FALSE;
			TASK:=1000;
		END_IF
		
	2000:
		IF ABB_Control_FB.qxPickedAGV THEN
			MAIN.qxABBExecutLamp:=FALSE;
			GVL.qxPickedfromAGV:=TRUE;
			ABB_Control_FB.qxPickAGV:=FALSE;
			ABB_Control_FB.ixPickAGV:=FALSE;
			TASK:=1000;
		END_IF
		
	2100:
		IF ABB_Control_FB.qxLeftAGV THEN
			MAIN.qxABBExecutLamp:=FALSE;
			GVL.qxPalletPlacedinAGV:=TRUE;
			ABB_Control_FB.qxLeaveAGV:=FALSE;
			ABB_Control_FB.ixLeaveAGV:=FALSE;
			TASK:=1000;
		END_IF
		
	2200:
			IF mxRP THEN
				GVL.BufferProducts.Storage1.Component:= 'Red Plate';
				GVL.BufferProducts.Storage1.Quatity:=2;
			ELSIF mxYP THEN
				GVL.BufferProducts.Storage1.Component:= 'Yellow Plate';
				GVL.BufferProducts.Storage1.Quatity:=2;
			ELSIF mxBP THEN
				GVL.BufferProducts.Storage1.Component:='Blue Plate';
				GVL.BufferProducts.Storage1.Quatity:=2;
			ELSIF mxRCy THEN
				GVL.BufferProducts.Storage1.Component:= 'Red Cylinder';
				GVL.BufferProducts.Storage1.Quatity:=4;
			ELSIF mxYCy THEN
				GVL.BufferProducts.Storage1.Component:= 'Yellow Cylinder';
				GVL.BufferProducts.Storage1.Quatity:=4;
			ELSIF mxBCy THEN
				GVL.BufferProducts.Storage1.Component:= 'Blue Cylinder';
				GVL.BufferProducts.Storage1.Quatity:=4;
			ELSIF mxROct THEN
				GVL.BufferProducts.Storage1.Component:= 'Red Octagon';
				GVL.BufferProducts.Storage1.Quatity:=4;
			ELSIF mxYOct THEN
				GVL.BufferProducts.Storage1.Component:= 'Yellow Octagon';
				GVL.BufferProducts.Storage1.Quatity:=4;
			ELSIF mxBOct THEN
				GVL.BufferProducts.Storage1.Component:= 'Blue Octagon';
				GVL.BufferProducts.Storage1.Quatity:=4;
			ELSIF mxIP THEN
				GVL.BufferProducts.Storage1.Component:='InvalidPart';
				GVL.BufferProducts.Storage1.Quatity:=0;
			END_IF
			TASK:=1000;
			
	2300:
			IF mxRP THEN
				GVL.BufferProducts.Storage1.Component:= 'Red Plate';
				GVL.BufferProducts.Storage1.Quatity:=2;
			ELSIF mxYP THEN
				GVL.BufferProducts.Storage1.Component:= 'Yellow Plate';
				GVL.BufferProducts.Storage1.Quatity:=2;
			ELSIF mxBP THEN
				GVL.BufferProducts.Storage1.Component:='Blue Plate';
				GVL.BufferProducts.Storage1.Quatity:=2;
			ELSIF mxRCy THEN
				GVL.BufferProducts.Storage1.Component:= 'Red Cylinder';
				GVL.BufferProducts.Storage1.Quatity:=4;
			ELSIF mxYCy THEN
				GVL.BufferProducts.Storage1.Component:= 'Yellow Cylinder';
				GVL.BufferProducts.Storage1.Quatity:=4;
			ELSIF mxBCy THEN
				GVL.BufferProducts.Storage1.Component:= 'Blue Cylinder';
				GVL.BufferProducts.Storage1.Quatity:=4;
			ELSIF mxROct THEN
				GVL.BufferProducts.Storage1.Component:= 'Red Octagon';
				GVL.BufferProducts.Storage1.Quatity:=4;
			ELSIF mxYOct THEN
				GVL.BufferProducts.Storage1.Component:= 'Yellow Octagon';
				GVL.BufferProducts.Storage1.Quatity:=4;
			ELSIF mxBOct THEN
				GVL.BufferProducts.Storage1.Component:= 'Blue Octagon';
				GVL.BufferProducts.Storage1.Quatity:=4;
			ELSIF mxIP THEN
				GVL.BufferProducts.Storage1.Component:='InvalidPart';
				GVL.BufferProducts.Storage1.Quatity:=0;
			END_IF
			TASK:=1000;
			
	2400:
			IF mxRP THEN
				GVL.BufferProducts.Storage1.Component:= 'Red Plate';
				GVL.BufferProducts.Storage1.Quatity:=2;
			ELSIF mxYP THEN
				GVL.BufferProducts.Storage1.Component:= 'Yellow Plate';
				GVL.BufferProducts.Storage1.Quatity:=2;
			ELSIF mxBP THEN
				GVL.BufferProducts.Storage1.Component:='Blue Plate';
				GVL.BufferProducts.Storage1.Quatity:=2;
			ELSIF mxRCy THEN
				GVL.BufferProducts.Storage1.Component:= 'Red Cylinder';
				GVL.BufferProducts.Storage1.Quatity:=4;
			ELSIF mxYCy THEN
				GVL.BufferProducts.Storage1.Component:= 'Yellow Cylinder';
				GVL.BufferProducts.Storage1.Quatity:=4;
			ELSIF mxBCy THEN
				GVL.BufferProducts.Storage1.Component:= 'Blue Cylinder';
				GVL.BufferProducts.Storage1.Quatity:=4;
			ELSIF mxROct THEN
				GVL.BufferProducts.Storage1.Component:= 'Red Octagon';
				GVL.BufferProducts.Storage1.Quatity:=4;
			ELSIF mxYOct THEN
				GVL.BufferProducts.Storage1.Component:= 'Yellow Octagon';
				GVL.BufferProducts.Storage1.Quatity:=4;
			ELSIF mxBOct THEN
				GVL.BufferProducts.Storage1.Component:= 'Blue Octagon';
				GVL.BufferProducts.Storage1.Quatity:=4;
			ELSIF mxIP THEN
				GVL.BufferProducts.Storage1.Component:='InvalidPart';
				GVL.BufferProducts.Storage1.Quatity:=0;
			END_IF
			TASK:=1000;
			
	2500:
		IF ABB_Control_FB.qxPickedTable THEN
			MAIN.qxABBExecutLamp:=FALSE;
			ABB_Control_FB.qxPickTable:=FALSE;
			ABB_Control_FB.ixPickTable:=FALSE;
			TASK:=1000;
		END_IF
		
	2600:
		IF ABB_Control_FB.qxLeftTable THEN
			MAIN.qxABBExecutLamp:=FALSE;
			ABB_Control_FB.qxLeaveTable:=FALSE;
			ABB_Control_FB.ixLeaveTable:=FALSE;
			TASK:=1000;
		END_IF
		
	2700:
				IF mxRCon THEN
					MAIN.qsContainer:='Red Container';
				ELSIF mxYCon THEN
					MAIN.qsContainer:='Yellow Container';
				ELSIF mxBCon THEN
					MAIN.qsContainer:='Blue Container';
				END_IF
				TASK:=1000;
				
	2800:
		IF ABB_Control_FB.mxCon_1_ATtableScan THEN
			IF GVL.ixInductiveSensorinTool THEN
				MAIN.mxPlateAvailable:=TRUE;
				TASK:=1000;
				ABB_Control_FB.ixScanPart1:=FALSE;
				MAIN.qxABBExecutLamp:=FALSE;
			ELSIF NOT GVL.ixInductiveSensorinTool THEN
				ABB_Control_FB.ixScanPart1:=FALSE;
				MAIN.qxABBExecutLamp:=FALSE;
				TASK:=1000;
			END_IF
		END_IF
		
	2900:
		IF ABB_Control_FB.mxCon_2_ATtableScan THEN
			IF GVL.ixInductiveSensorinTool THEN
				MAIN.mxCylinderAvailable:=TRUE;
				TASK:=1000;
				ABB_Control_FB.ixScanPart2:=FALSE;
				MAIN.qxABBExecutLamp:=FALSE;
			ELSIF NOT GVL.ixInductiveSensorinTool THEN
				ABB_Control_FB.ixScanPart2:=FALSE;
				MAIN.qxABBExecutLamp:=FALSE;
				TASK:=1000;
			END_IF
		END_IF
		
	3000:
		IF ABB_Control_FB.mxCon_2_ATtableScan THEN
			IF GVL.ixInductiveSensorinTool THEN
				MAIN.mxOctagonAvailable:=TRUE;
				TASK:=1000;
				ABB_Control_FB.ixScanPart3:=FALSE;
				MAIN.qxABBExecutLamp:=FALSE;
			ELSIF NOT GVL.ixInductiveSensorinTool THEN
				ABB_Control_FB.ixScanPart3:=FALSE;
				MAIN.qxABBExecutLamp:=FALSE;
				TASK:=1000;
			END_IF
		END_IF
		
	3100:
		IF ABB_Control_FB.mxAsse_1_done THEN
			mxPart1:=TRUE;
			ABB_Control_FB.ixAssemble1:=FALSE;
			MAIN.qxABBExecutLamp:=FALSE;
			TASK:=1000;
		END_IF
		
	3200:
		IF ABB_Control_FB.mxAsse_2_done THEN
			mxPart2:=TRUE;
			ABB_Control_FB.ixAssemble2:=FALSE;
			MAIN.qxABBExecutLamp:=FALSE;
			TASK:=1000;
		END_IF
		
	3300:
		IF ABB_Control_FB.mxAsse_3_done THEN
			mxPart3:=TRUE;
			ABB_Control_FB.ixAssemble3:=FALSE;
			MAIN.qxABBExecutLamp:=FALSE;
			TASK:=1000;
		END_IF
		
	3400:
		IF NOT MAIN.mxPlateAvailable AND mxPart1 THEN
			IF MAIN.qsContainer='Red Container' THEN
				GVL.qsOrderFornextAssembly:='Red Plate';
			ELSIF MAIN.qsContainer='Yellow Container' THEN
				GVL.qsOrderFornextAssembly:='Yellow Plate';
			ELSIF MAIN.qsContainer='Blue Container' THEN
				GVL.qsOrderFornextAssembly:='Blue Plate';
			ELSE
				TASK:=3500;
			END_IF
		END_IF
		
	3500:
		IF mxPart2 OR MAIN.mxCylinderAvailable THEN
			mxSLOT1:=TRUE;
			TASK:=3600;
		ELSE
			mxSLOT1:=FALSE;
			TASK:=3600;
		END_IF
		
	3600:
	 	IF mxPART3 OR MAIN.mxOctagonAvailable THEN
		 	mxSLOT2:=TRUE;
		 	TASK:=3800;
		ELSE
			mxSLOT2:=FALSE;
			TASK:=3800;
	 	END_IF
	 
	3800:
		IF MAIN.qsContainer='Yellow Container' THEN
			IF mxSLOT1 AND mxSLOT2 THEN 
					   gvl.qsOrderFornextAssembly:='Assembled Product';
					   TASK:=3900;
					   ELSIF mxSLOT1 AND NOT mxSLOT2 THEN 
						   gvl.qsOrderFornextAssembly:='Yellow Octagon';
					    TASK:=3900;
					   ELSIF NOT mxSLOT1 AND mxSLOT2 THEN 
						   gvl.qsOrderFornextAssembly:='Yellow Cylinder';
					    TASk:=3900;
					   ELSIF NOT mxSLOT1 AND NOT mxSLOT2 THEN
						  gvl.qsOrderFornextAssembly:='Yellow Cylinder';
					    TASK:=3900; 
				   END_IF
				   
		ELSIF MAIN.qsContainer='Red Container' THEN
			IF mxSLOT1 AND mxSLOT2 THEN 
					   gvl.qsOrderFornextAssembly:='Assembled Product';
					   TASK:=3900;
					   ELSIF mxSLOT1 AND NOT mxSLOT2 THEN 
						   gvl.qsOrderFornextAssembly:='Red Octagon';
					    TASK:=3900;
					   ELSIF NOT mxSLOT1 AND mxSLOT2 THEN 
						   gvl.qsOrderFornextAssembly:='Red Cylinder';
					    TASk:=3900;
					   ELSIF NOT mxSLOT1 AND NOT mxSLOT2 THEN
						  gvl.qsOrderFornextAssembly:='Red Cylinder';
					    TASK:=3900; 
				   END_IF
				   
		ELSIF MAIN.qsContainer='Blue Container' THEN
			IF mxSLOT1 AND mxSLOT2 THEN 
					   gvl.qsOrderFornextAssembly:='Assembled Product';
					   TASK:=3900;
					   ELSIF mxSLOT1 AND NOT mxSLOT2 THEN 
						   gvl.qsOrderFornextAssembly:='Blue Octagon';
					    TASK:=3900;
					   ELSIF NOT mxSLOT1 AND mxSLOT2 THEN 
						   gvl.qsOrderFornextAssembly:='Blue Cylinder';
					    TASk:=3900;
					   ELSIF NOT mxSLOT1 AND NOT mxSLOT2 THEN
						  gvl.qsOrderFornextAssembly:='Blue Cylinder';
					    TASK:=3900; 
				   END_IF
		
		END_IF
		
	3900:
		IF ABB_Control_FB.ixFinishOrder THEN
			ABB_Control_FB.mxAsse_1_done:=FALSE;
			ABB_Control_FB.mxAsse_2_done:=FALSE;
			ABB_Control_FB.mxAsse_3_done:=FALSE;
			GVL.qsOrderFornextAssembly:='0';
			TASK:=1000;
		END_IF
		
	2001: // Emergency Stop
		ABB_Control_FB.qxScanBuffer_1:=FALSE;
		ABB_Control_FB.qxScanBuffer_2:=FALSE;
		ABB_Control_FB.qxScanBuffer_3:=FALSE;
		ABB_Control_FB.ixGoTo_AGV:=FALSE;
		ABB_Control_FB.qxCon1:=FALSE;
		ABB_Control_FB.qxCon2:=FALSE;
		ABB_Control_FB.qxCon3:=FALSE;
		ABB_Control_FB.qxPart_1_Assemble:=FALSE;
		ABB_Control_FB.qxPart_2_Assemble:=FALSE;
		ABB_Control_FB.qxPart_3_Assemble:=FALSE;
		ABB_Control_FB.qxAssemblyDone:=FALSE;
	 
	
END_CASE

END_FUNCTION_BLOCK

(* stored: Version 1.1.0.1, ProductVersion 3.1.4024.12
   POU Scanner_FB: Id {ca46032a-69db-43ab-b12e-fff7cb39dbfa}, SpecialFunc None *)
